{attribute 'qualified_only'}
{attribute 'strict'}
TYPE StateEnum :
(
  undefined,
  idle,
  busy,
  error
);
END_TYPE

(* stored: Version 1.1.0.1, ProductVersion 3.1.4024.9
   DUT StateEnum: Id {1b401aa7-ce7a-4de0-8dde-e86175fd1d75} *)
